{attribute 'linkalways'} 
{attribute 'no_explicit_call' := 'This FB is a CLASS and must be accessed using methods or properties'}
{attribute 'enable_dynamic_creation'}
FUNCTION_BLOCK _ETcVnFlipAxis EXTENDS EnumDatatypeBase
VAR
	localData : ETcVnFlipAxis;
	activeData : REFERENCE TO ETcVnFlipAxis;
	enumBaseDatatype : _INT(localData);
END_VAR

METHOD PRIVATE AddLocalEnumeration
VAR_INPUT
	Enumeration : T_MAXSTRING;
	Value : ETcVnFlipAxis;
END_VAR
AddEnumeration(Enumeration, Value);
END_METHOD

PROPERTY PUBLIC Address : PVOID
GET
Address := ADR(activeData);
END_GET
END_PROPERTY

METHOD PUBLIC ClearReference
VAR_INPUT
END_VAR
activeData REF= localData;
SetBaseDatatypeReference();
END_METHOD

METHOD PUBLIC Clone : I_Datatype
VAR
    pClone : POINTER TO _ETcVnFlipAxis;
END_VAR
pClone := __NEW(_ETcVnFlipAxis(InitialValue := Value));
Clone := pClone^;
END_METHOD

METHOD FB_init : BOOL
VAR_INPUT
	bInitRetains : BOOL; // if TRUE, the retain variables are initialized (warm start / cold start)
	bInCopyCode : BOOL;  // if TRUE, the instance afterwards gets moved into the copy code (online change)
	InitialValue : ETcVnFlipAxis;
END_VAR
localData := InitialValue;
AddBaseDatatype(enumBaseDatatype);
ClearReference();

AddLocalEnumeration('TCVN_FA_XY', ETcVnFlipAxis.TCVN_FA_XY);
AddLocalEnumeration('TCVN_FA_X', ETcVnFlipAxis.TCVN_FA_X);
AddLocalEnumeration('TCVN_FA_Y', ETcVnFlipAxis.TCVN_FA_Y);
END_METHOD

PROPERTY PUBLIC Identifier : T_MAXSTRING
GET
Identifier := 'ETcVnFlipAxis';
END_GET
END_PROPERTY

METHOD IsEnumeratorValueEqual : BOOL
VAR_INPUT
	Enumerator : I_KeyValueForwardEnumerator;
END_VAR
VAR
	storedValue : ETcVnFlipAxis;
END_VAR
IF NOT Enumerator.TryGet(storedValue) THEN
	RETURN;
END_IF

IsEnumeratorValueEqual := storedValue = activeData;
END_METHOD

METHOD PUBLIC MakeReferenceTo
VAR_INPUT
	ReferenceTarget : REFERENCE TO ETcVnFlipAxis;
END_VAR
activeData REF= ReferenceTarget;
SetBaseDatatypeReference();
END_METHOD

METHOD PROTECTED SetBaseDatatypeReference
VAR_INPUT
END_VAR
enumBaseDatatype.MakeReferenceTo(activeData);
END_METHOD

PROPERTY PUBLIC Size : UDINT
GET
Size := SIZEOF(activeData);
END_GET
END_PROPERTY

METHOD TryMakeReferenceTo : BOOL
VAR_INPUT
	Target : I_Datatype;
END_VAR
VAR
	targetAsEnum : I_EnumDatatype;
	pTargetData : POINTER TO ETcVnFlipAxis;
END_VAR
IF NOT Target.TryResolveAsEnumDatatype(targetAsEnum) THEN
	RETURN;
END_IF

IF targetAsEnum.Identifier <> Identifier THEN
	RETURN;
END_IF

pTargetData := Target.Address;
activeData REF= pTargetData^;
SetBaseDatatypeReference();
TryMakeReferenceTo := TRUE;
END_METHOD

PROPERTY PUBLIC Value : ETcVnFlipAxis
GET
Value := activeData;
END_GET
SET
activeData := Value;
END_SET
END_PROPERTY

END_FUNCTION_BLOCK

(* stored: Version 1.1.0.1, ProductVersion 3.1.4024.12
   POU _ETcVnFlipAxis: Id {c6227475-ba2b-0f63-0fbd-5ef1b55e4837}, SpecialFunc None
   Folder Constructor: Id {bec19af7-c488-0719-2170-996a781fda0a}
   Folder Private: Id {131cc083-1d16-0a99-2e6d-79f848b11990}
   Folder Protected: Id {4827eb1b-c1e4-0227-0866-ab2c04f0f9b0}
   Method AddLocalEnumeration: Id {89272682-ba9a-08e8-2754-b23b38576dbd}
   Property Address: Id {a6c5bebb-8d67-0b59-0c29-4ded7292d7d9}
   Get Get: Id {9f8172f2-a265-0d7a-2ac3-5b9d03fbc6ef}
   Method ClearReference: Id {cffe9a52-1a19-0321-02d9-2989619ae05b}
   Method Clone: Id {2012daed-fc94-0cab-1572-b116514ab3a8}
   Method FB_init: Id {e4f8cdc1-0562-03cd-1db3-d66f79227dc6}
   Property Identifier: Id {36bcd99c-fcc5-0ef5-1d70-bc23e43da643}
   Get Get: Id {4f13a932-dd36-0d6c-1445-d91b2e41b840}
   Method IsEnumeratorValueEqual: Id {fd9dfd47-9297-0e9c-0600-4306d2618656}
   Method MakeReferenceTo: Id {6ed1c7e6-3825-0260-1ad3-af3236e7431b}
   Method SetBaseDatatypeReference: Id {56414470-879c-08da-287b-5a0973e1e693}
   Property Size: Id {46134a94-2ce1-083e-19f9-d28e4b62f7af}
   Get Get: Id {1e1c2c64-1a28-0db0-3c4a-3810761cf147}
   Method TryMakeReferenceTo: Id {19e87bd4-9061-0435-18f9-de75138a63cd}
   Property Value: Id {fcec4666-6a55-0a48-19a9-e3b57def03fa}
   Get Get: Id {96c19c76-66d5-08e5-3060-b04734c8ed48}
   Set Set: Id {ee0ed036-b7fa-08b3-23ca-165ef28a2126} *)
